// TIA Portal V17 export
// export: Created 2025-03-05T08:01:38.1195353Z, ExportSetting WithDefaults, DisplayName Totally Integrated Automation Portal, DisplayVersion V17 Update 8, DisplayName TIA Portal Openness, DisplayVersion V17 Update 8, DisplayName TIA Portal Version Control Interface, DisplayVersion V17, DisplayName SINAMICS Startdrive Advanced, DisplayVersion V17 SP2, DisplayName SINAMICS Startdrive G110M, G120, G120C, G120D, G120P, G115D, DisplayVersion V17 SP2, DisplayName SINAMICS Startdrive G130, G150, S120, S150, SINAMICS MV, S210, DisplayVersion V17 SP2, DisplayName STEP 7 Professional, DisplayVersion V17 Update 8, DisplayName SINUMERIK ONE STEP 7 Toolbox, DisplayVersion V17 Update 12, DisplayName SINUMERIK 840D sl STEP 7 Toolbox, DisplayVersion V17 Update 12, DisplayName STEP 7 Safety, DisplayVersion V17 Update 6, DisplayName WinCC Advanced, DisplayVersion V17 Update 8
FUNCTION "FC7210_PRODUCTION" : Void   // FC7210, LAD
{ S7_Optimized_Access := 'FALSE' }
AUTHOR : ETXETAR
VERSION : 1.0
// stored: AutoNumber false, IsIECCheckEnabled false, SetENOAutomatically false, UDAEnableTagReadback false
   VAR_TEMP
      FIXTURE_1_ENABLE_COUNT : Bool;   // FIXTURE 1 ENABLE COUNT
      FIXTURE_2_ENABLE_COUNT : Bool;   // FIXTURE 2 ENABLE COUNT
      PHD_ARM_1_ENABLE_COUNT : Bool;   // PHD ARM 1 ENABLE COUNT
      PHD_ARM_2_ENABLE_COUNT : Bool;   // PHD ARM 2 ENABLE COUNT
   END_VAR
BEGIN

REGION Network 1: FIXTURE 1 ENABLE COUNT / ENABLE FIXTURE 1 COUNT
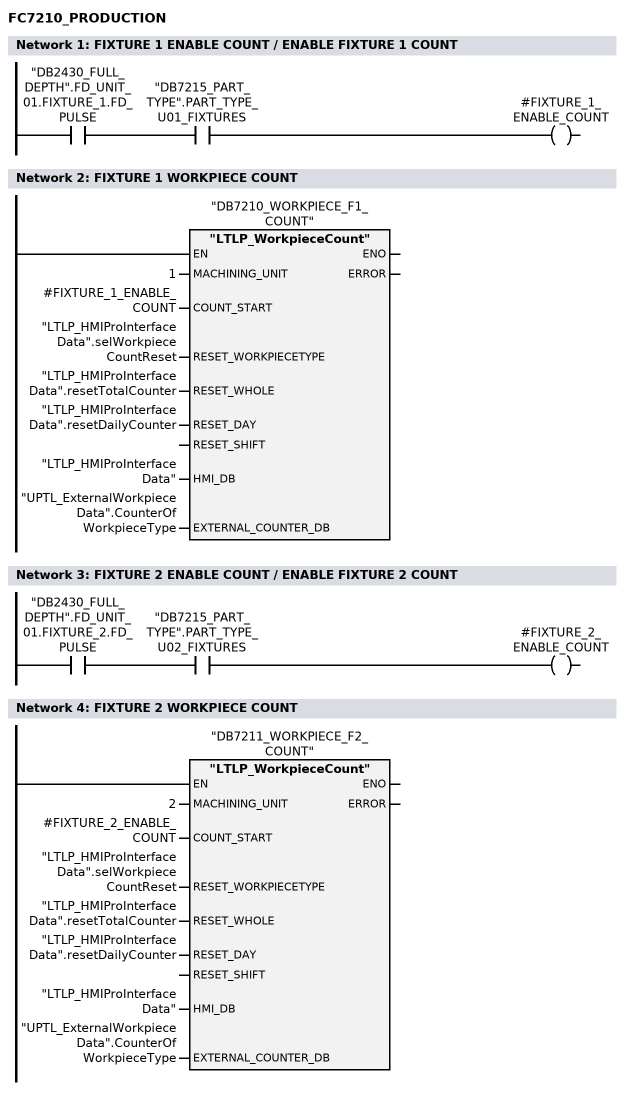
   RUNG wire#powerrail
      Contact( "DB2430_FULL_DEPTH".FD_UNIT_01.FIXTURE_1.FD_PULSE )
      Contact( "DB7215_PART_TYPE".PART_TYPE_U01_FIXTURES )
      Coil( #FIXTURE_1_ENABLE_COUNT )
   END_RUNG
   // the same network as SCL:
   #FIXTURE_1_ENABLE_COUNT := "DB2430_FULL_DEPTH".FD_UNIT_01.FIXTURE_1.FD_PULSE AND "DB7215_PART_TYPE".PART_TYPE_U01_FIXTURES;
END_REGION

REGION Network 2: FIXTURE 1 WORKPIECE COUNT
   RUNG wire#powerrail
      "DB7210_WORKPIECE_F1_COUNT"(MACHINING_UNIT := 1, COUNT_START := #FIXTURE_1_ENABLE_COUNT, RESET_WORKPIECETYPE := "LTLP_HMIProInterfaceData".selWorkpieceCountReset, RESET_WHOLE := "LTLP_HMIProInterfaceData".resetTotalCounter, RESET_DAY := "LTLP_HMIProInterfaceData".resetDailyCounter, RESET_SHIFT :=, HMI_DB := "LTLP_HMIProInterfaceData", EXTERNAL_COUNTER_DB := "UPTL_ExternalWorkpieceData".CounterOfWorkpieceType, ERROR =>)
   END_RUNG
   // the same network as SCL:
   "DB7210_WORKPIECE_F1_COUNT"(MACHINING_UNIT := 1,   // "LTLP_WorkpieceCount"
                           COUNT_START := #FIXTURE_1_ENABLE_COUNT,
                           RESET_WORKPIECETYPE := "LTLP_HMIProInterfaceData".selWorkpieceCountReset,
                           RESET_WHOLE := "LTLP_HMIProInterfaceData".resetTotalCounter,
                           RESET_DAY := "LTLP_HMIProInterfaceData".resetDailyCounter,
                           HMI_DB := "LTLP_HMIProInterfaceData",
                           EXTERNAL_COUNTER_DB := "UPTL_ExternalWorkpieceData".CounterOfWorkpieceType);
END_REGION

REGION Network 3: FIXTURE 2 ENABLE COUNT / ENABLE FIXTURE 2 COUNT
   RUNG wire#powerrail
      Contact( "DB2430_FULL_DEPTH".FD_UNIT_01.FIXTURE_2.FD_PULSE )
      Contact( "DB7215_PART_TYPE".PART_TYPE_U02_FIXTURES )
      Coil( #FIXTURE_2_ENABLE_COUNT )
   END_RUNG
   // the same network as SCL:
   #FIXTURE_2_ENABLE_COUNT := "DB2430_FULL_DEPTH".FD_UNIT_01.FIXTURE_2.FD_PULSE AND "DB7215_PART_TYPE".PART_TYPE_U02_FIXTURES;
END_REGION

REGION Network 4: FIXTURE 2 WORKPIECE COUNT
   RUNG wire#powerrail
      "DB7211_WORKPIECE_F2_COUNT"(MACHINING_UNIT := 2, COUNT_START := #FIXTURE_2_ENABLE_COUNT, RESET_WORKPIECETYPE := "LTLP_HMIProInterfaceData".selWorkpieceCountReset, RESET_WHOLE := "LTLP_HMIProInterfaceData".resetTotalCounter, RESET_DAY := "LTLP_HMIProInterfaceData".resetDailyCounter, RESET_SHIFT :=, HMI_DB := "LTLP_HMIProInterfaceData", EXTERNAL_COUNTER_DB := "UPTL_ExternalWorkpieceData".CounterOfWorkpieceType, ERROR =>)
   END_RUNG
   // the same network as SCL:
   "DB7211_WORKPIECE_F2_COUNT"(MACHINING_UNIT := 2,   // "LTLP_WorkpieceCount"
                           COUNT_START := #FIXTURE_2_ENABLE_COUNT,
                           RESET_WORKPIECETYPE := "LTLP_HMIProInterfaceData".selWorkpieceCountReset,
                           RESET_WHOLE := "LTLP_HMIProInterfaceData".resetTotalCounter,
                           RESET_DAY := "LTLP_HMIProInterfaceData".resetDailyCounter,
                           HMI_DB := "LTLP_HMIProInterfaceData",
                           EXTERNAL_COUNTER_DB := "UPTL_ExternalWorkpieceData".CounterOfWorkpieceType);
END_REGION
END_FUNCTION
